FUNCTION_BLOCK FB_Extract_Num_Mes
// extract phone number from the received message
VAR_INPUT
    InMessage     : STRING(255);
END_VAR
VAR_OUTPUT
    OutDataEntry  :ST_SMSDataSetEntry_Read;
END_VAR
VAR
    ChaineTmp     : STRING(255);
    Num           : STRING(255);
    Pos           : INT;
    Pos1          : INT;
    Pos2          : INT;
    Pos3          : INT;    
	Offset		: INT ; 
END_VAR

//+CMGR: "REC UNREAD","+33776039883",,"18/04/19,18:25:44+08"$R$NBonjour je m'appelle henry$R$N 50
Pos:=FIND(InMessage,',"');
chaineTmp:=MID(InMessage,LEN(InMessage)-21,POS+2);
Pos1:=FIND(chaineTmp,'",,');
Num:=MID(chaineTmp,Pos1-1,1);
Pos3:= FIND(Num,'+');
OutDataEntry.Num:= SEL(Pos3= 0 ,Num ,CONCAT(STR1:= CstPhoneIndicator_G, STR2:= Num) );
Pos2:=FIND(InMessage,'$R$N');
Offset := FIND(MID(InMessage,LEN(InMessage)-Pos2,Pos2+2),'$R$N') ;


OutDataEntry.Message:=MID(InMessage,Offset-1,Pos2+2);//OutDataEntry.Message:=MID(InMessage,LEN(InMessage)-Pos2-3,LEN(InMessage));	// OutDataEntry.Message:=MID(InMessage,LEN(InMessage)-Pos2-3,Pso2+2);

END_FUNCTION_BLOCK

(* stored: Version 1.1.0.1, ProductVersion 3.1.4024.6
   POU FB_Extract_Num_Mes: Id {27b567bf-402a-447f-96df-a2e65a2a70a2}, SpecialFunc None *)
